FUNCTION_BLOCK FB_DO EXTENDS FB_Basic
VAR_INPUT
	bValue		: BOOL;

END_VAR
VAR_OUTPUT
END_VAR
VAR
// HW
	{attribute 'OPC.UA.DA':='1'}
	{attribute 'OPC.UA.DA.Access' := '1'}
	{attribute 'OPC.UA.DA.Description' := 'Output I/O signal'}
	{attribute 'OPC.UA.DA.StructuredType' := '0'}
	Output AT %Q* : BOOL;		// Value to IO module
	State AT %I* : WORD := 8;	// State from Ethercat module

END_VAR


// Run parent FB
SUPER^();

METHOD PROTECTED M_AutoMode : BOOL
VAR_INPUT
END_VAR
// Digital outputs automatic mode
// Executed from parent FB_Basic

rAutoValue := BOOL_TO_LREAL(bValue);

IF (P_bEnable) THEN
	rActualValue := rAutoValue;
ELSE
	rActualValue := 0.0;
END_IF
END_METHOD

METHOD PROTECTED M_ErrorHandling : BOOL
VAR_INPUT
END_VAR
// Error handling
IF (bCmdEnable) THEN
	IF (NOT P_bManualMode) THEN
		// Hardware errors
		IF (NOT F_ECat_OK(State)) THEN
			// EtherCAT state
			bStaError := TRUE;
			eStaErrorID := E_ComponentErrors.HW_ECat_Not_OP;
		END_IF
	END_IF
	
ELSE
	bStaError := FALSE;
	bStaWarning := FALSE;
	eStaErrorID := E_ComponentErrors.OK;

END_IF
END_METHOD

METHOD PROTECTED M_Init : BOOL
VAR_INPUT
END_VAR
// Init

bCmdEnable := TRUE;
bInitDone := TRUE;
END_METHOD

METHOD PROTECTED M_ManualMode : BOOL
VAR_INPUT
END_VAR
// Digital outputs manual mode
// Executed from parent FB_Basic

rManualValue := LIMIT(0, rManualValue, 1);

IF (P_bEnable) THEN
	rActualValue := rManualValue;
ELSE
	rActualValue := 0.0;
END_IF
END_METHOD

METHOD PROTECTED M_Run : BOOL
VAR_INPUT
END_VAR
// Analog inputs run
// Executed from parent FB_Basic

// Update IO 

Output := LREAL_TO_BOOL(rActualValue);
END_METHOD

END_FUNCTION_BLOCK

(* stored: Version 1.1.0.1, ProductVersion 3.1.4024.2
   POU FB_DO: Id {dcfed493-6bc4-4f58-bf17-8d52ea5d5d6c}, SpecialFunc None
   Method M_AutoMode: Id {5e77ac08-bc02-468e-87bd-27616ccd25a8}
   Method M_ErrorHandling: Id {97c577e9-a47f-4b2f-90c8-5bac06877bfe}
   Method M_Init: Id {3d396bf6-6dd0-4b60-a6bd-bd3b30c044f6}
   Method M_ManualMode: Id {b8023084-ef59-4f5c-99a5-d4942205aa09}
   Method M_Run: Id {3c81795b-99ec-44cc-8c08-1eab2a4f33c3} *)
